# EPICS autosave request: soft_iocs/galil_DMC/iocBoot/iocgalil_DMC_E06_08/DMC_Positions.req
$(P)$(M1).DVAL
$(P)$(M2).DVAL
$(P)$(M3).DVAL
$(P)$(M4).DVAL
$(P)$(M5).DVAL
$(P)$(M6).DVAL
$(P)$(M7).DVAL
$(P)$(M8).DVAL
